// TIA Portal V16 export
// export: Created 2023-01-04T15:44:09.8920418Z, ExportSetting WithDefaults, DisplayName Totally Integrated Automation Portal, DisplayVersion V16, DisplayName TIA Portal Version Control Interface, DisplayVersion V16, DisplayName TIA Portal Openness, DisplayVersion V16, DisplayName STEP 7 Professional, DisplayVersion V16, DisplayName STEP 7 Safety, DisplayVersion V16, DisplayName WinCC Advanced, DisplayVersion V16
VAR_GLOBAL   // PLC tag table "Default tag table"
   FIC_B102 AT %IW64 : Int;
   LIC_B101 AT %IW66 : Int;
   PS1_RFID_Station AT %I0.0 : Bool;   // PS-Proximity Switch
   PS2_Filling_Station AT %I0.1 : Bool;
   PS3_Quality_Station AT %I0.2 : Bool;
   PS4_End_of_Conveyor AT %I0.3 : Bool;
   T01_Low_Level AT %I0.4 : Bool;
   T01_High_Level AT %I0.5 : Bool;
   T01_Outlet AT %Q0.1 : Bool;
   T02_Outlet AT %Q0.2 : Bool;
   Outlet_Pump_Motor AT %Q0.3 : Bool;
   Conveyor_Motor AT %Q0.0 : Bool;
   NTRG_06 AT %M5.5 : Bool;
   NTRG_09 AT %M5.6 : Bool;
   NTRG_099 AT %M5.7 : Bool;
   PTRG10 AT %M6.0 : Bool;
   PTRIG999 AT %M6.1 : Bool;
   PTRIG998 AT %M6.2 : Bool;
   PTRIG888 AT %M6.3 : Bool;
   ptrig141 AT %M6.4 : Bool;
   ptrig142 AT %M6.5 : Bool;
   ptrig143 AT %M6.6 : Bool;
END_VAR
